% RSLogix 500 project P5_IVANOVSKI_M.RSS, saved by version 8.30.00.16 %
PROJECT "UNTITLED"    % processor: Bul.1763 MicroLogix 1100 Series B %

PROGRAM FILES
  LAD 2   7 rungs

DATA FILES
  O0 OUTPUT  4 elements
  I1 INPUT  6 elements
  S2 STATUS  66 elements
  B3 BINARY  1 elements
  T4 TIMER  2 elements
  C5 COUNTER  1 elements
  R6 CONTROL  1 elements
  N7 INTEGER  1 elements
  F8 FLOAT  3 elements

LADDER 2
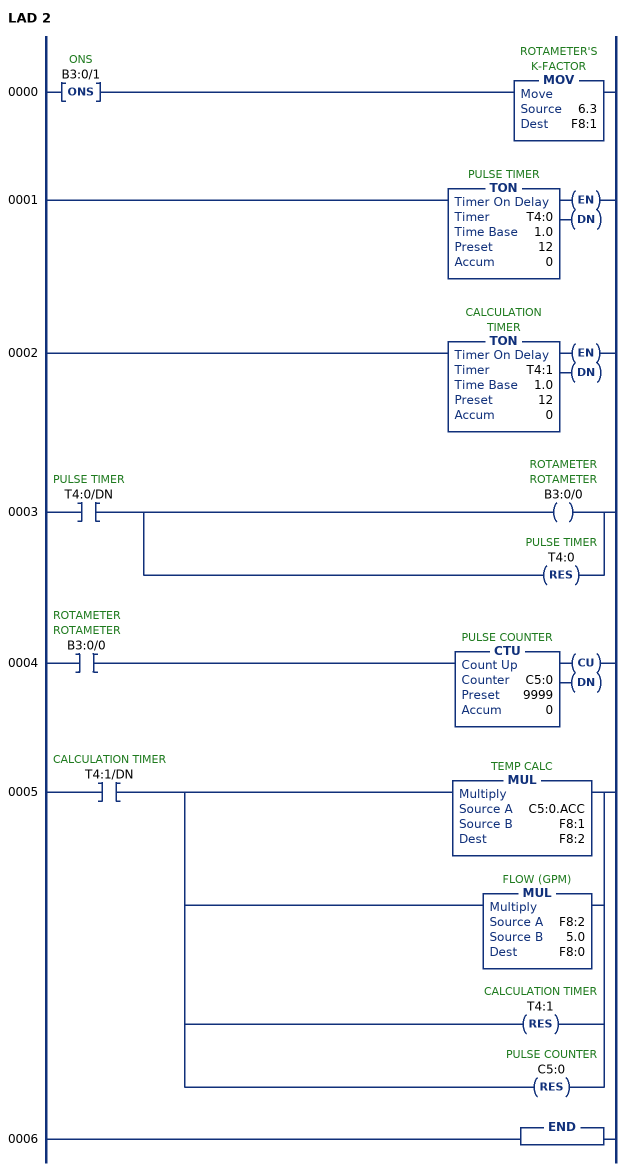
% Rung: 0 %
SOR ONS B3:0/1 MOV 6.3 F8:1 EOR
%   B3:0/1  "ONS" %
%   F8:1  "ROTAMETER'S K-FACTOR" %
% Rung: 1 %
SOR TON T4:0 1.0 12 0 EOR
%   T4:0  "PULSE TIMER" %
% Rung: 2 %
SOR TON T4:1 1.0 12 0 EOR
%   T4:1  "CALCULATION TIMER" %
% Rung: 3 %
SOR XIC T4:0/DN BST OTE B3:0/0 NXB RES T4:0 BND EOR
%   T4:0/DN  "PULSE TIMER" %
%   B3:0/0  ROTAMETER  "ROTAMETER" %
%   T4:0  "PULSE TIMER" %
% Rung: 4 %
SOR XIC B3:0/0 CTU C5:0 9999 0 EOR
%   B3:0/0  ROTAMETER  "ROTAMETER" %
%   C5:0  "PULSE COUNTER" %
% Rung: 5 %
SOR XIC T4:1/DN BST MUL C5:0.ACC F8:1 F8:2 NXB MUL F8:2 5.0 F8:0 NXB RES T4:1 NXB RES C5:0 BND EOR
%   T4:1/DN  "CALCULATION TIMER" %
%   C5:0.ACC  "TEMP CALC" %
%   F8:1  "ROTAMETER'S K-FACTOR" %
%   F8:2  "TEMP CALC" %
%   F8:0  "FLOW (GPM)" %
%   T4:1  "CALCULATION TIMER" %
%   C5:0  "PULSE COUNTER" %
% Rung: 6 %
SOR END EOR

DATA TABLE (non-zero values as saved)
DATA T4
% .PRE .ACC %
% T4:0 % 12 0
% T4:1 % 12 0
DATA C5
% .PRE .ACC %
% C5:0 % 9999 0
